SYSTEM test
  (* Version 1.0, 2023-07-01, franz *)
  DEVICE FORTE_PC : FORTE_PC(MGR_ID := C_00)
    {SET_ATTRIBUTE(Profile, HOLOBLOC)}
    RESOURCE EMB_RES : EMB_RES
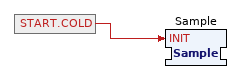
      SUBAPPS
        Sample : Sample;
      END_SUBAPPS
      EVENT_CONNECTIONS
        START.COLD TO Sample.INIT;
      END_CONNECTIONS
    END_RESOURCE
  END_DEVICE
  SEGMENTS
    Ethernet : Ethernet;
  END_SEGMENTS
  LINKS
    FORTE_PC => Ethernet;
  END_LINKS
END_SYSTEM
